(* PLC project , CODESYS CODESYS V3.5 SP8 Patch 4 *)
(* stored: creationDateTime 2018-11-14T08:45:48.2560871, modificationDateTime 2018-11-14T08:45:35.8305333 *)

VAR_GLOBAL  (* LogLibBasic *)
  GlobalLogBufferHandle : LogBufferHandle;
  GlobalTick : UDINT;
END_VAR

FUNCTION CreateGlobalBufferHandle : BOOL
VAR_INPUT
    BufferAddress: POINTER TO BYTE;
    BufferSize: DINT;
END_VAR
VAR
END_VAR

            CreateBufferHandle(BufferAddress, BufferSize, GlobalLogBufferHandle);

          
END_FUNCTION

FUNCTION LogBool : BOOL
VAR_INPUT
    Group: BYTE;
    Id: BYTE;
    Channel: UINT;
    Value: BOOL;
END_VAR
VAR
END_VAR

            IF Group > 0 OR Id > 0 THEN
    IF Channel < 256 THEN
        EvtGr8Id8Ch8Tick32Bool8(Group, Id, UINT_TO_BYTE(Channel), GlobalTick, Value, GlobalLogBufferHandle);
    ELSE
        EvtGr8Id8Ch16Tick32Bool8(Group, Id, Channel, GlobalTick, Value, GlobalLogBufferHandle);
    END_IF
ELSIF Channel < 256 THEN
    EvtCh8Tick32Bool8(UINT_TO_BYTE(Channel), GlobalTick, Value, GlobalLogBufferHandle);
ELSE
    EvtCh16Tick32Bool8(Channel, GlobalTick, Value, GlobalLogBufferHandle);
END_IF

          
END_FUNCTION

FUNCTION LogInt : BOOL
VAR_INPUT
    Group: BYTE;
    Id: BYTE;
    Channel: UINT;
    Value: INT;
END_VAR
VAR
END_VAR

            IF Group > 0 OR Id > 0 THEN
    IF Channel < 256 THEN
        EvtGr8Id8Ch8Tick32Int16(Group, Id, UINT_TO_BYTE(Channel), GlobalTick, Value, GlobalLogBufferHandle);
    ELSE
        EvtGr8Id8Ch16Tick32Int16(Group, Id, Channel, GlobalTick, Value, GlobalLogBufferHandle);
    END_IF
ELSIF Channel < 256 THEN
    EvtCh8Tick32Int16(UINT_TO_BYTE(Channel), GlobalTick, Value, GlobalLogBufferHandle);
ELSE
    EvtCh16Tick32Int16(Channel, GlobalTick, Value, GlobalLogBufferHandle);
END_IF

          
END_FUNCTION

FUNCTION LogDInt : BOOL
VAR_INPUT
    Group: BYTE;
    Id: BYTE;
    Channel: UINT;
    Value: DINT;
END_VAR
VAR
END_VAR

            IF Group > 0 OR Id > 0 THEN
    IF Channel < 256 THEN
        EvtGr8Id8Ch8Tick32Int32(Group, Id, UINT_TO_BYTE(Channel), GlobalTick, Value, GlobalLogBufferHandle);
    ELSE
        EvtGr8Id8Ch16Tick32Int32(Group, Id, Channel, GlobalTick, Value, GlobalLogBufferHandle);
    END_IF
ELSIF Channel < 256 THEN
    EvtCh8Tick32Int32(UINT_TO_BYTE(Channel), GlobalTick, Value, GlobalLogBufferHandle);
ELSE
    EvtCh16Tick32Int32(Channel, GlobalTick, Value, GlobalLogBufferHandle);
END_IF

          
END_FUNCTION

FUNCTION LogUDInt : BOOL
VAR_INPUT
    Group: BYTE;
    Id: BYTE;
    Channel: UINT;
    Value: UDINT;
END_VAR
VAR
END_VAR

            IF Group > 0 OR Id > 0 THEN
    IF Channel < 256 THEN
        EvtGr8Id8Ch8Tick32UInt32(Group, Id, UINT_TO_BYTE(Channel), GlobalTick, Value, GlobalLogBufferHandle);
    ELSE
        EvtGr8Id8Ch16Tick32UInt32(Group, Id, Channel, GlobalTick, Value, GlobalLogBufferHandle);
    END_IF
ELSIF Channel < 256 THEN
    EvtCh8Tick32UInt32(UINT_TO_BYTE(Channel), GlobalTick, Value, GlobalLogBufferHandle);
ELSE
    EvtCh16Tick32UInt32(Channel, GlobalTick, Value, GlobalLogBufferHandle);
END_IF

          
END_FUNCTION

FUNCTION LogReal : BOOL
VAR_INPUT
    Group: BYTE;
    Id: BYTE;
    Channel: UINT;
    Value: REAL;
END_VAR
VAR
END_VAR

            IF Group > 0 OR Id > 0 THEN
    IF Channel < 256 THEN
        EvtGr8Id8Ch8Tick32Real32(Group, Id, UINT_TO_BYTE(Channel), GlobalTick, Value, GlobalLogBufferHandle);
    ELSE
        EvtGr8Id8Ch16Tick32Real32(Group, Id, Channel, GlobalTick, Value, GlobalLogBufferHandle);
    END_IF
ELSIF Channel < 256 THEN
    EvtCh8Tick32Real32(UINT_TO_BYTE(Channel), GlobalTick, Value, GlobalLogBufferHandle);
ELSE
    EvtCh16Tick32Real32(Channel, GlobalTick, Value, GlobalLogBufferHandle);
END_IF

          
END_FUNCTION

FUNCTION LogLReal : BOOL
VAR_INPUT
    Group: BYTE;
    Id: BYTE;
    Channel: UINT;
    Value: LREAL;
END_VAR
VAR
END_VAR

            IF Group > 0 OR Id > 0 THEN
    IF Channel < 256 THEN
        EvtGr8Id8Ch8Tick32Real64(Group, Id, UINT_TO_BYTE(Channel), GlobalTick, Value, GlobalLogBufferHandle);
    ELSE
        EvtGr8Id8Ch16Tick32Real64(Group, Id, Channel, GlobalTick, Value, GlobalLogBufferHandle);
    END_IF
ELSIF Channel < 256 THEN
    EvtCh8Tick32Real64(UINT_TO_BYTE(Channel), GlobalTick, Value, GlobalLogBufferHandle);
ELSE
    EvtCh16Tick32Real64(Channel, GlobalTick, Value, GlobalLogBufferHandle);
END_IF

          
END_FUNCTION

FUNCTION MonitorBool : BOOL
VAR_INPUT
    Group: BYTE;
    Id: BYTE;
    Channel: UINT;
    Value: BOOL;
END_VAR
VAR_IN_OUT
    Data: BOOL;
END_VAR
VAR
END_VAR

            IF Value <> Data THEN
    IF Group > 0 OR Id > 0 THEN
        IF Channel < 256 THEN
            EvtGr8Id8Ch8Tick32Bool8(Group, Id, UINT_TO_BYTE(Channel), GlobalTick, Value, GlobalLogBufferHandle);
        ELSE
            EvtGr8Id8Ch16Tick32Bool8(Group, Id, Channel, GlobalTick, Value, GlobalLogBufferHandle);
        END_IF
    ELSIF Channel < 256 THEN
        EvtCh8Tick32Bool8(UINT_TO_BYTE(Channel), GlobalTick, Value, GlobalLogBufferHandle);
    ELSE
        EvtCh16Tick32Bool8(Channel, GlobalTick, Value, GlobalLogBufferHandle);
    END_IF
    Data := Value;
END_IF

          
END_FUNCTION

FUNCTION MonitorInt : BOOL
VAR_INPUT
    Group: BYTE;
    Id: BYTE;
    Channel: UINT;
    Value: INT;
END_VAR
VAR_IN_OUT
    Data: INT;
END_VAR
VAR
END_VAR

            IF Value <> Data THEN
    IF Group > 0 OR Id > 0 THEN
        IF Channel < 256 THEN
            EvtGr8Id8Ch8Tick32Int16(Group, Id, UINT_TO_BYTE(Channel), GlobalTick, Value, GlobalLogBufferHandle);
        ELSE
            EvtGr8Id8Ch16Tick32Int16(Group, Id, Channel, GlobalTick, Value, GlobalLogBufferHandle);
        END_IF
    ELSIF Channel < 256 THEN
        EvtCh8Tick32Int16(UINT_TO_BYTE(Channel), GlobalTick, Value, GlobalLogBufferHandle);
    ELSE
        EvtCh16Tick32Int16(Channel, GlobalTick, Value, GlobalLogBufferHandle);
    END_IF
    Data := Value;
END_IF

          
END_FUNCTION

FUNCTION MonitorDInt : BOOL
VAR_INPUT
    Group: BYTE;
    Id: BYTE;
    Channel: UINT;
    Value: DINT;
END_VAR
VAR_IN_OUT
    Data: DINT;
END_VAR
VAR
END_VAR

            IF Value <> Data THEN
    IF Group > 0 OR Id > 0 THEN
        IF Channel < 256 THEN
            EvtGr8Id8Ch8Tick32Int32(Group, Id, UINT_TO_BYTE(Channel), GlobalTick, Value, GlobalLogBufferHandle);
        ELSE
            EvtGr8Id8Ch16Tick32Int32(Group, Id, Channel, GlobalTick, Value, GlobalLogBufferHandle);
        END_IF
    ELSIF Channel < 256 THEN
        EvtCh8Tick32Int32(UINT_TO_BYTE(Channel), GlobalTick, Value, GlobalLogBufferHandle);
    ELSE
        EvtCh16Tick32Int32(Channel, GlobalTick, Value, GlobalLogBufferHandle);
    END_IF
    Data := Value;
END_IF

          
END_FUNCTION

FUNCTION MonitorUDInt : BOOL
VAR_INPUT
    Group: BYTE;
    Id: BYTE;
    Channel: UINT;
    Value: UDINT;
END_VAR
VAR_IN_OUT
    Data: UDINT;
END_VAR
VAR
END_VAR

            IF Value <> Data THEN
    IF Group > 0 OR Id > 0 THEN
        IF Channel < 256 THEN
            EvtGr8Id8Ch8Tick32UInt32(Group, Id, UINT_TO_BYTE(Channel), GlobalTick, Value, GlobalLogBufferHandle);
        ELSE
            EvtGr8Id8Ch16Tick32UInt32(Group, Id, Channel, GlobalTick, Value, GlobalLogBufferHandle);
        END_IF
    ELSIF Channel < 256 THEN
        EvtCh8Tick32UInt32(UINT_TO_BYTE(Channel), GlobalTick, Value, GlobalLogBufferHandle);
    ELSE
        EvtCh16Tick32UInt32(Channel, GlobalTick, Value, GlobalLogBufferHandle);
    END_IF
    Data := Value;
END_IF

          
END_FUNCTION

FUNCTION MonitorReal : BOOL
VAR_INPUT
    Group: BYTE;
    Id: BYTE;
    Channel: UINT;
    Value: REAL;
END_VAR
VAR_IN_OUT
    Data: REAL;
END_VAR
VAR
END_VAR

            IF Value <> Data THEN
    IF Group > 0 OR Id > 0 THEN
        IF Channel < 256 THEN
            EvtGr8Id8Ch8Tick32Real32(Group, Id, UINT_TO_BYTE(Channel), GlobalTick, Value, GlobalLogBufferHandle);
        ELSE
            EvtGr8Id8Ch16Tick32Real32(Group, Id, Channel, GlobalTick, Value, GlobalLogBufferHandle);
        END_IF
    ELSIF Channel < 256 THEN
        EvtCh8Tick32Real32(UINT_TO_BYTE(Channel), GlobalTick, Value, GlobalLogBufferHandle);
    ELSE
        EvtCh16Tick32Real32(Channel, GlobalTick, Value, GlobalLogBufferHandle);
    END_IF
    Data := Value;
END_IF

          
END_FUNCTION

FUNCTION MonitorLReal : BOOL
VAR_INPUT
    Group: BYTE;
    Id: BYTE;
    Channel: UINT;
    Value: LREAL;
END_VAR
VAR_IN_OUT
    Data: LREAL;
END_VAR
VAR
END_VAR

            IF Value <> Data THEN
    IF Group > 0 OR Id > 0 THEN
        IF Channel < 256 THEN
            EvtGr8Id8Ch8Tick32Real64(Group, Id, UINT_TO_BYTE(Channel), GlobalTick, Value, GlobalLogBufferHandle);
        ELSE
            EvtGr8Id8Ch16Tick32Real64(Group, Id, Channel, GlobalTick, Value, GlobalLogBufferHandle);
        END_IF
    ELSIF Channel < 256 THEN
        EvtCh8Tick32Real64(UINT_TO_BYTE(Channel), GlobalTick, Value, GlobalLogBufferHandle);
    ELSE
        EvtCh16Tick32Real64(Channel, GlobalTick, Value, GlobalLogBufferHandle);
    END_IF
    Data := Value;
END_IF

          
END_FUNCTION
